{attribute addProperty BoxType "EL2912-0000-0016"}
{attribute addProperty Id "OutputsOutputs_2D8468E2162"}
{attribute addProperty CRC "1749617362"}
{attribute addProperty SizeInBites "16"}
{attribute addProperty SizeInBytes "2"}
TYPE Module_2_FSOUT_68490AD2 :
STRUCT
	{attribute addProperty Name "Outputs"}
	Outputs  : Outputs_2D8468E2;
END_STRUCT
END_TYPE

(* stored: Version 1.2.0.0, ProductVersion 3.1.4024.9
   DUT Module_2_FSOUT_68490AD2: Id {627a37ea-f1f9-4c41-af57-3c21bcf5e350} *)
